// TIA Portal V20 export
ORGANIZATION_BLOCK "Main"   // OB1, LAD, ProgramCycle
TITLE = "Main Program Sweep (Cycle)"
{ S7_Optimized_Access := 'TRUE' }
// stored: SetENOAutomatically false
   VAR_INPUT
      Initial_Call : Bool;   // Initial call of this OB
      Remanence : Bool;   // =True, if remanent data are available
   END_VAR
   VAR_TEMP
      tst : Bool;
      tst_ergebnis : Bool;
   END_VAR
BEGIN

REGION Network 1: Testchange
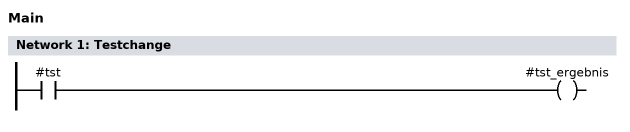
   RUNG wire#powerrail
      Contact( #tst )
      Coil( #tst_ergebnis )
   END_RUNG
   // the same network as SCL:
   #tst_ergebnis := #tst;
END_REGION
END_ORGANIZATION_BLOCK
